FUNCTION_BLOCK BatteryModelClient (* Client FB for delegating battery model simulations to an external server. *)
  (* Standard: 61499-2 *)
  (* Version 1.0, 2017-06-18, Marc Jakobi, HTW Berlin *)
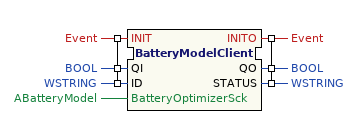
  EVENT_INPUT
    INIT WITH QI, ID; (* Initialization Request *)
  END_EVENT
  EVENT_OUTPUT
    INITO WITH QO, STATUS; (* Initialization Confirm *)
  END_EVENT
  VAR_INPUT
    QI : BOOL; (* Input event qualifier *)
    ID : WSTRING; (* Connection Identifier *)
  END_VAR
  VAR_OUTPUT
    QO : BOOL; (* Output event qualifier *)
    STATUS : WSTRING; (* Service Status *)
  END_VAR
  SOCKETS
    BatteryOptimizerSck : ABatteryModel; (* Link to BatteryOptimizer *)
  END_SOCKETS
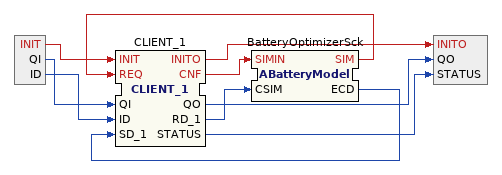
  FBS
    CLIENT_1 : CLIENT_1;
  END_FBS
  EVENT_CONNECTIONS
    INIT TO CLIENT_1.INIT;
    CLIENT_1.INITO TO INITO;
    BatteryOptimizerSck.SIM TO CLIENT_1.REQ;
    CLIENT_1.CNF TO BatteryOptimizerSck.SIMIN;
  END_CONNECTIONS
  DATA_CONNECTIONS
    QI TO CLIENT_1.QI;
    ID TO CLIENT_1.ID;
    CLIENT_1.QO TO QO;
    BatteryOptimizerSck.ECD TO CLIENT_1.SD_1;
    CLIENT_1.RD_1 TO BatteryOptimizerSck.CSIM;
    CLIENT_1.STATUS TO STATUS;
  END_CONNECTIONS
END_FUNCTION_BLOCK
